// TIA Portal V20 export
DATA_BLOCK "EeMonitor"   // DB61
TITLE = EeMonitor
AUTHOR : SICAR
FAMILY : DB
// Globale EEM Informationen / Global EEM Information
// stored: InstanceOfName LSicar_typeEemDataHmi, InstanceOfType UDT
"LSicar_typeEemDataHmi"
   // VAR
   //    measurePointIndex : USInt;
   //    measConfiguration { ExternalWritable := 'False'} : EnS_EEm_typeMeasConfig;
   //    measOperationHmi { ExternalWritable := 'False'} : EnS_EEm_typeMeasOperation;
   //    work { ExternalWritable := 'False'} : "LSicar_typeEnMeterWorkHmi";
   // END_VAR
BEGIN
END_DATA_BLOCK
